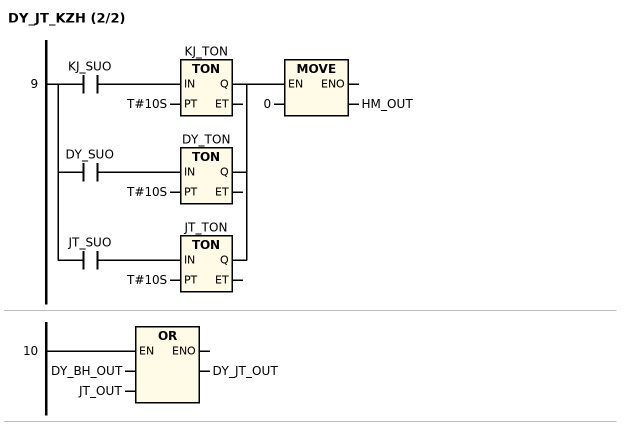
[picture p72: DY_JT_KZH (LD)]
_LD_ (* Ladder Diagram *)
NETWORK 1 (* 电源保护延时控制 *)
	{ [DY_BH_IN] | [DY_BH_OUT] } - [TD_TON_IN] - [/DY_FW] - [/JT_OUT] - [/REST] --- (DY_BH_OUT)
NETWORK 2
	[DY_BH_OUT] - [/DY_BH_IN] - DY_OPEN:YANSHI_OPEN(EN_IN: *, TIME_IN: MUL(DY_FW_SET, 60), ET_OUT => DY_BH_ET) --- (DY_FW)
NETWORK 3
	*
		EN --- LIMIT(5, DY_FW_SET, 60) => DY_FW_SET
NETWORK 4 (* 急停控制 *)
	[JT_IN] --- (JT_OUT)
NETWORK 5
	KJ_R:R_TRIG(CLK: *)
		EN --- MOVE(1) => HM_OUT
NETWORK 6
	[DY_BH_OUT] - DY_R:R_TRIG(CLK: *)
		EN --- MOVE(2) => HM_OUT
NETWORK 7
	[JT_OUT] - JT_R:R_TRIG(CLK: *)
		EN --- MOVE(4) => HM_OUT
NETWORK 8
	*
		EN --- EQ(HM_OUT, 1) => KJ_SUO
		EN --- EQ(HM_OUT, 2) => DY_SUO
		EN --- EQ(HM_OUT, 4) => JT_SUO
NETWORK 9
	{ [KJ_SUO] - KJ_TON:TON(IN: *, PT: T#10S) | [DY_SUO] - DY_TON:TON(IN: *, PT: T#10S) | [JT_SUO] - JT_TON:TON(IN: *, PT: T#10S) }
		EN --- MOVE(0) => HM_OUT
NETWORK 10
	*
		EN --- OR(DY_BH_OUT, JT_OUT) => DY_JT_OUT
_END_LD_
(* the same logic as Structured Text *)
(* Network 1: 电源保护延时控制 *)
DY_BH_OUT := (DY_BH_IN OR DY_BH_OUT) AND TD_TON_IN AND NOT DY_FW AND NOT JT_OUT AND NOT REST;
(* Network 2 *)
DY_OPEN(EN_IN := DY_BH_OUT AND NOT DY_BH_IN, TIME_IN := DY_FW_SET * 60);
DY_BH_ET := DY_OPEN.ET_OUT;
DY_FW := DY_OPEN.OUT;
(* Network 3 *)
DY_FW_SET := LIMIT(5, DY_FW_SET, 60);
(* Network 4: 急停控制 *)
JT_OUT := JT_IN;
(* Network 5 *)
KJ_R(CLK := TRUE);
IF KJ_R.Q THEN
	HM_OUT := 1;
END_IF;
(* Network 6 *)
DY_R(CLK := DY_BH_OUT);
IF DY_R.Q THEN
	HM_OUT := 2;
END_IF;
(* Network 7 *)
JT_R(CLK := JT_OUT);
IF JT_R.Q THEN
	HM_OUT := 4;
END_IF;
(* Network 8 *)
KJ_SUO := HM_OUT = 1;
DY_SUO := HM_OUT = 2;
JT_SUO := HM_OUT = 4;
(* Network 9 *)
KJ_TON(IN := KJ_SUO, PT := T#10S);
DY_TON(IN := DY_SUO, PT := T#10S);
JT_TON(IN := JT_SUO, PT := T#10S);
IF KJ_TON.Q OR DY_TON.Q OR JT_TON.Q THEN
	HM_OUT := 0;
END_IF;
(* Network 10 *)
DY_JT_OUT := DY_BH_OUT OR JT_OUT;
END_FUNCTION_BLOCK

(* POU MONI_LIANG_PW, LD *)
FUNCTION_BLOCK MONI_LIANG_PW
VAR_INPUT
	DY_IN: WORD;
	XZH_IN: INT;


	XH_IN: BOOL;


	ALA_L_T_IN: INT;
	ALA_L_T_YSH: WORD;

	ALA_H_T_IN: INT;
	ALA_H_T_YSH: WORD;


	REST: BOOL;
	JJQ_K: INT;
	JJQ_G: INT;
	YSH_IN: WORD;
END_VAR
VAR_OUTPUT
	MONI_OUT: INT;
	ALA_L_OUT: BOOL;
	ALA_H_OUT: BOOL;
	ALA_T_ET: WORD;
	PW_ZHT: WORD;
	JJQ_OUT: BOOL;
	JZ_OUT: BOOL;
END_VAR
VAR








	ALA_H_KA_0: BOOL;
	ALA_H_KA: BOOL;
	ALA_H_TON: YANSHI_OPEN;
	ALA_L_KA_0: BOOL;
	ALA_L_TON: YANSHI_OPEN;
	ALA_L_KA: BOOL;
	ALA_H_T_ET: WORD;
	ALA_L_T_ET: WORD;



	HEX_ENGIN: HEX_ENGIN;
	K1: BOOL;
	G1: BOOL;
	KJ: BOOL;
	YANSHI_OPEN: YANSHI_OPEN;
	TOF: TOF;
	YANSHI_CLOSE: YANSHI_CLOSE;
END_VAR
VAR_IN_OUT
END_VAR
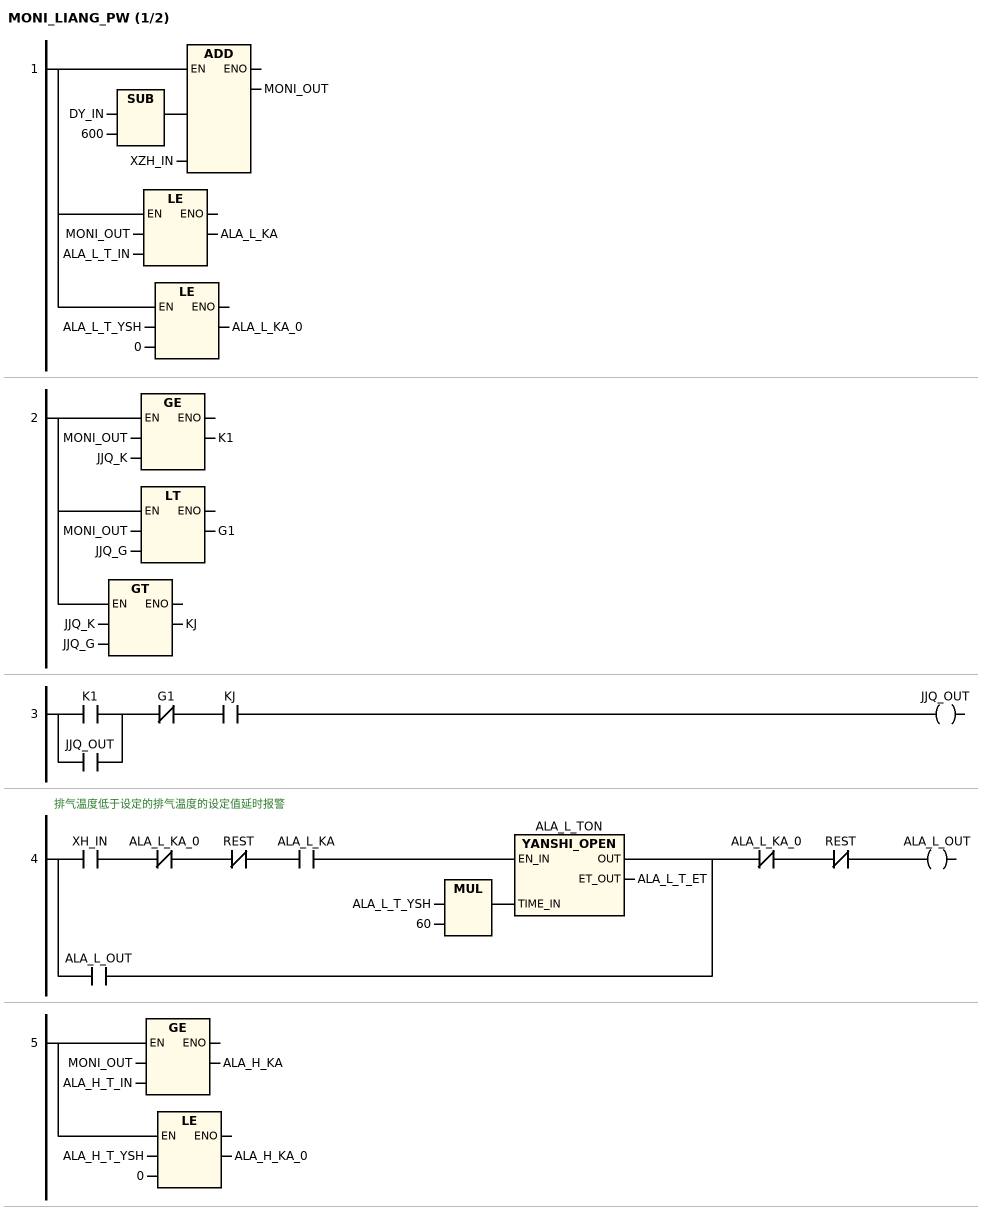
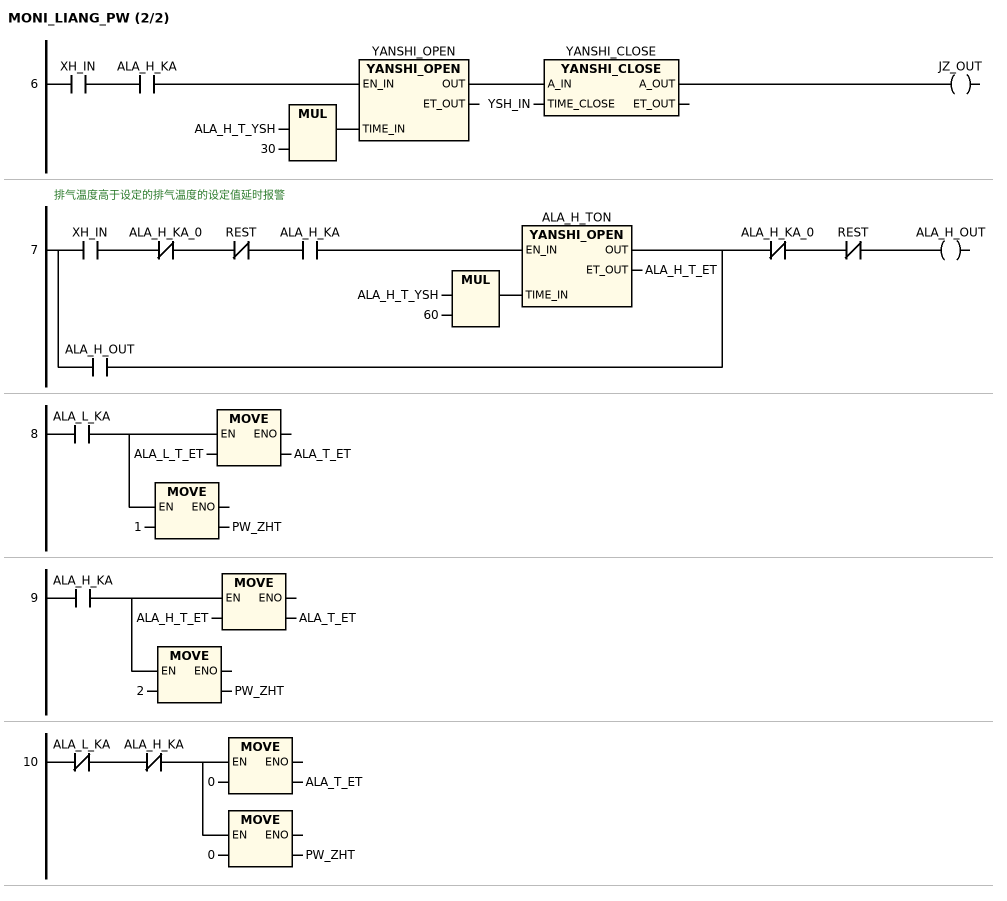
_LD_ (* Ladder Diagram *)
NETWORK 1
	*
		EN --- ADD(SUB(DY_IN, 600), XZH_IN) => MONI_OUT
		EN --- LE(MONI_OUT, ALA_L_T_IN) => ALA_L_KA
		EN --- LE(ALA_L_T_YSH, 0) => ALA_L_KA_0
NETWORK 2
	*
		EN --- GE(MONI_OUT, JJQ_K) => K1
		EN --- LT(MONI_OUT, JJQ_G) => G1
		EN --- GT(JJQ_K, JJQ_G) => KJ
NETWORK 3
	{ [K1] | [JJQ_OUT] } - [/G1] - [KJ] --- (JJQ_OUT)
NETWORK 4 (* 排气温度低于设定的排气温度的设定值延时报警 *)
	{ [XH_IN] - [/ALA_L_KA_0] - [/REST] - [ALA_L_KA] - ALA_L_TON:YANSHI_OPEN(EN_IN: *, TIME_IN: MUL(ALA_L_T_YSH, 60), ET_OUT => ALA_L_T_ET) | [ALA_L_OUT] } - [/ALA_L_KA_0] - [/REST] --- (ALA_L_OUT)
NETWORK 5
	*
		EN --- GE(MONI_OUT, ALA_H_T_IN) => ALA_H_KA
		EN --- LE(ALA_H_T_YSH, 0) => ALA_H_KA_0
NETWORK 6
	[XH_IN] - [ALA_H_KA] - YANSHI_OPEN:YANSHI_OPEN(EN_IN: *, TIME_IN: MUL(ALA_H_T_YSH, 30)) - YANSHI_CLOSE:YANSHI_CLOSE(A_IN: *, TIME_CLOSE: YSH_IN) --- (JZ_OUT)
NETWORK 7 (* 排气温度高于设定的排气温度的设定值延时报警 *)
	{ [XH_IN] - [/ALA_H_KA_0] - [/REST] - [ALA_H_KA] - ALA_H_TON:YANSHI_OPEN(EN_IN: *, TIME_IN: MUL(ALA_H_T_YSH, 60), ET_OUT => ALA_H_T_ET) | [ALA_H_OUT] } - [/ALA_H_KA_0] - [/REST] --- (ALA_H_OUT)
NETWORK 8
	[ALA_L_KA]
		EN --- MOVE(ALA_L_T_ET) => ALA_T_ET
		EN --- MOVE(1) => PW_ZHT
NETWORK 9
	[ALA_H_KA]
		EN --- MOVE(ALA_H_T_ET) => ALA_T_ET
		EN --- MOVE(2) => PW_ZHT
NETWORK 10
	[/ALA_L_KA] - [/ALA_H_KA]
		EN --- MOVE(0) => ALA_T_ET
		EN --- MOVE(0) => PW_ZHT
_END_LD_
(* the same logic as Structured Text *)
(* Network 1 *)
MONI_OUT := (DY_IN - 600) + XZH_IN;
ALA_L_KA := MONI_OUT <= ALA_L_T_IN;
ALA_L_KA_0 := ALA_L_T_YSH <= 0;
(* Network 2 *)
K1 := MONI_OUT >= JJQ_K;
G1 := MONI_OUT < JJQ_G;
KJ := JJQ_K > JJQ_G;
(* Network 3 *)
JJQ_OUT := (K1 OR JJQ_OUT) AND NOT G1 AND KJ;
(* Network 4: 排气温度低于设定的排气温度的设定值延时报警 *)
ALA_L_TON(EN_IN := XH_IN AND NOT ALA_L_KA_0 AND NOT REST AND ALA_L_KA, TIME_IN := ALA_L_T_YSH * 60);
ALA_L_T_ET := ALA_L_TON.ET_OUT;
ALA_L_OUT := (ALA_L_TON.OUT OR ALA_L_OUT) AND NOT ALA_L_KA_0 AND NOT REST;
(* Network 5 *)
ALA_H_KA := MONI_OUT >= ALA_H_T_IN;
ALA_H_KA_0 := ALA_H_T_YSH <= 0;
(* Network 6 *)
YANSHI_OPEN(EN_IN := XH_IN AND ALA_H_KA, TIME_IN := ALA_H_T_YSH * 30);
YANSHI_CLOSE(A_IN := YANSHI_OPEN.OUT, TIME_CLOSE := YSH_IN);
JZ_OUT := YANSHI_CLOSE.A_OUT;
(* Network 7: 排气温度高于设定的排气温度的设定值延时报警 *)
ALA_H_TON(EN_IN := XH_IN AND NOT ALA_H_KA_0 AND NOT REST AND ALA_H_KA, TIME_IN := ALA_H_T_YSH * 60);
ALA_H_T_ET := ALA_H_TON.ET_OUT;
ALA_H_OUT := (ALA_H_TON.OUT OR ALA_H_OUT) AND NOT ALA_H_KA_0 AND NOT REST;
(* Network 8 *)
IF ALA_L_KA THEN
	ALA_T_ET := ALA_L_T_ET;
	PW_ZHT := 1;
END_IF;
(* Network 9 *)
IF ALA_H_KA THEN
	ALA_T_ET := ALA_H_T_ET;
	PW_ZHT := 2;
END_IF;
(* Network 10 *)
IF NOT ALA_L_KA AND NOT ALA_H_KA THEN
	ALA_T_ET := 0;
	PW_ZHT := 0;
END_IF;
END_FUNCTION_BLOCK

(* POU OPEN_KJ, LD *)
FUNCTION_BLOCK OPEN_KJ
VAR_INPUT
	H_IN: WORD;
	M_IN: WORD;
	KG_IN: BOOL;
	H_OPEN_1_IN: WORD;
	M_OPEN_1_IN: WORD;
	H_CLOSE_1_IN: WORD;
       M_CLOSE_1_IN: WORD;
	H_OPEN_2_IN: WORD;
	M_OPEN_2_IN: WORD;
	H_CLOSE_2_IN: WORD;
       M_CLOSE_2_IN: WORD;
	H_OPEN_3_IN: WORD;
	M_OPEN_3_IN: WORD;
	H_CLOSE_3_IN: WORD;
       M_CLOSE_3_IN: WORD;
END_VAR
VAR_OUTPUT
	KG_OUT: BOOL;
	KZH_OUT: BOOL;
END_VAR
VAR
	OPEN_1_KA: BOOL;
	CLOSE_1_KA: BOOL;
	OPEN_2_KA: BOOL;
	CLOSE_2_KA: BOOL;
	CLOSE_3_KA: BOOL;
	OPEN_3_KA: BOOL;

	KZH_2_OUT: BOOL;
	KZH_3_OUT: BOOL;
	KZH_1_OUT: BOOL;
	AN_K: AN_NIU;
END_VAR
VAR_IN_OUT

END_VAR
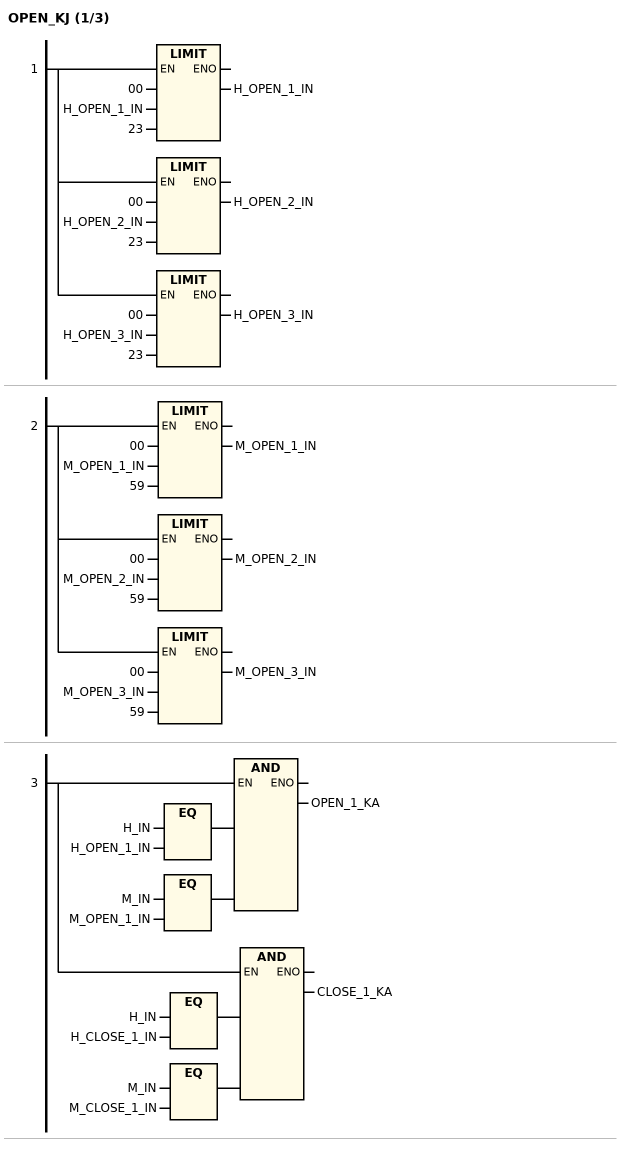
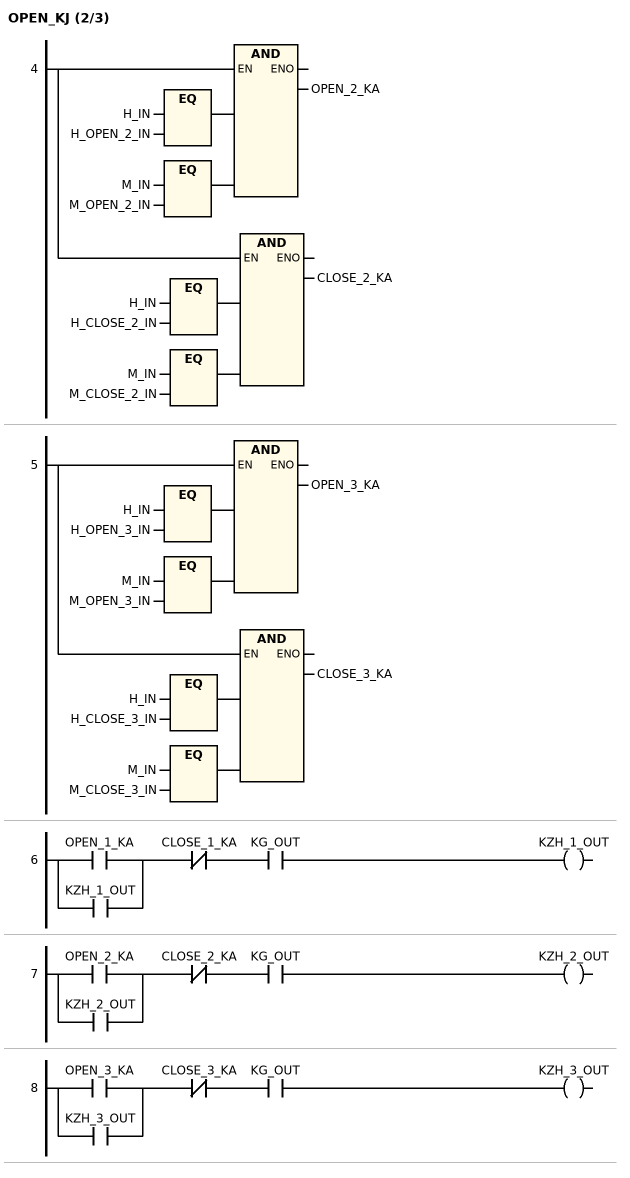
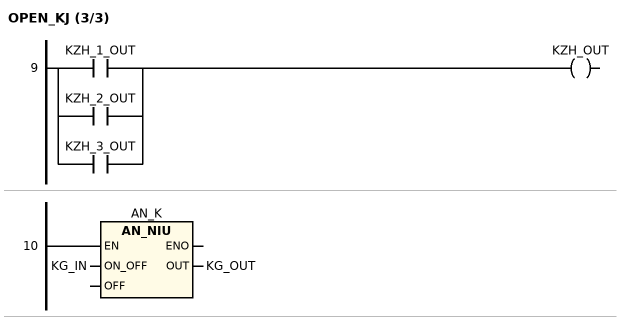
_LD_ (* Ladder Diagram *)
NETWORK 1
	*
		EN --- LIMIT(00, H_OPEN_1_IN, 23) => H_OPEN_1_IN
		EN --- LIMIT(00, H_OPEN_2_IN, 23) => H_OPEN_2_IN
		EN --- LIMIT(00, H_OPEN_3_IN, 23) => H_OPEN_3_IN
NETWORK 2
	*
		EN --- LIMIT(00, M_OPEN_1_IN, 59) => M_OPEN_1_IN
		EN --- LIMIT(00, M_OPEN_2_IN, 59) => M_OPEN_2_IN
		EN --- LIMIT(00, M_OPEN_3_IN, 59) => M_OPEN_3_IN
NETWORK 3
	*
		EN --- AND(EQ(H_IN, H_OPEN_1_IN), EQ(M_IN, M_OPEN_1_IN)) => OPEN_1_KA
		EN --- AND(EQ(H_IN, H_CLOSE_1_IN), EQ(M_IN, M_CLOSE_1_IN)) => CLOSE_1_KA
NETWORK 4
	*
		EN --- AND(EQ(H_IN, H_OPEN_2_IN), EQ(M_IN, M_OPEN_2_IN)) => OPEN_2_KA
		EN --- AND(EQ(H_IN, H_CLOSE_2_IN), EQ(M_IN, M_CLOSE_2_IN)) => CLOSE_2_KA
NETWORK 5
	*
		EN --- AND(EQ(H_IN, H_OPEN_3_IN), EQ(M_IN, M_OPEN_3_IN)) => OPEN_3_KA
		EN --- AND(EQ(H_IN, H_CLOSE_3_IN), EQ(M_IN, M_CLOSE_3_IN)) => CLOSE_3_KA
NETWORK 6
	{ [OPEN_1_KA] | [KZH_1_OUT] } - [/CLOSE_1_KA] - [KG_OUT] --- (KZH_1_OUT)
NETWORK 7
	{ [OPEN_2_KA] | [KZH_2_OUT] } - [/CLOSE_2_KA] - [KG_OUT] --- (KZH_2_OUT)
NETWORK 8
	{ [OPEN_3_KA] | [KZH_3_OUT] } - [/CLOSE_3_KA] - [KG_OUT] --- (KZH_3_OUT)
NETWORK 9
	{ [KZH_1_OUT] | [KZH_2_OUT] | [KZH_3_OUT] } --- (KZH_OUT)
NETWORK 10
	*
		EN --- AN_K:AN_NIU(ON_OFF: KG_IN, OFF: ) => KG_OUT
_END_LD_
(* the same logic as Structured Text *)
(* Network 1 *)
H_OPEN_1_IN := LIMIT(00, H_OPEN_1_IN, 23);
H_OPEN_2_IN := LIMIT(00, H_OPEN_2_IN, 23);
H_OPEN_3_IN := LIMIT(00, H_OPEN_3_IN, 23);
(* Network 2 *)
M_OPEN_1_IN := LIMIT(00, M_OPEN_1_IN, 59);
M_OPEN_2_IN := LIMIT(00, M_OPEN_2_IN, 59);
M_OPEN_3_IN := LIMIT(00, M_OPEN_3_IN, 59);
(* Network 3 *)
OPEN_1_KA := (H_IN = H_OPEN_1_IN) AND (M_IN = M_OPEN_1_IN);
CLOSE_1_KA := (H_IN = H_CLOSE_1_IN) AND (M_IN = M_CLOSE_1_IN);
(* Network 4 *)
OPEN_2_KA := (H_IN = H_OPEN_2_IN) AND (M_IN = M_OPEN_2_IN);
CLOSE_2_KA := (H_IN = H_CLOSE_2_IN) AND (M_IN = M_CLOSE_2_IN);
(* Network 5 *)
OPEN_3_KA := (H_IN = H_OPEN_3_IN) AND (M_IN = M_OPEN_3_IN);
CLOSE_3_KA := (H_IN = H_CLOSE_3_IN) AND (M_IN = M_CLOSE_3_IN);
(* Network 6 *)
KZH_1_OUT := (OPEN_1_KA OR KZH_1_OUT) AND NOT CLOSE_1_KA AND KG_OUT;
(* Network 7 *)
KZH_2_OUT := (OPEN_2_KA OR KZH_2_OUT) AND NOT CLOSE_2_KA AND KG_OUT;
(* Network 8 *)
KZH_3_OUT := (OPEN_3_KA OR KZH_3_OUT) AND NOT CLOSE_3_KA AND KG_OUT;
(* Network 9 *)
KZH_OUT := KZH_1_OUT OR KZH_2_OUT OR KZH_3_OUT;
(* Network 10: see the listing above *)
END_FUNCTION_BLOCK

(* POU DEF_YUNSUAN, LD *)
FUNCTION_BLOCK DEF_YUNSUAN
VAR_INPUT
	COOL_1_M: DWORD;
	COOL_2_M: DWORD;
	COOL_3_M: DWORD;
	COOL_4_M: DWORD;
	COOL_5_M: DWORD;
	COOL_6_M: DWORD;
	COOL_7_M: DWORD;
	COOL_8_M: DWORD;
	COOL_9_M: DWORD;
	COOL_10_M: DWORD;
	COOL_11_M: DWORD;
	COOL_12_M: DWORD;
	COOL_13_M: DWORD;
	COOL_14_M: DWORD;
	DD_1_IN: BOOL;
	DD_2_IN: BOOL;
	DD_3_IN: BOOL;
	DD_4_IN: BOOL;
	DD_5_IN: BOOL;
	DD_6_IN: BOOL;
	DD_7_IN: BOOL;
	DD_8_IN: BOOL;
	DD_9_IN: BOOL;
	DD_10_IN: BOOL;
	DD_11_IN: BOOL;
	DD_12_IN: BOOL;
	DD_13_IN: BOOL;
	DD_14_IN: BOOL;
	KSH_SET: WORD;

END_VAR
VAR_OUTPUT
	DEF_1_ZD: BOOL;
	DEF_2_ZD: BOOL;
	DEF_3_ZD: BOOL;
	DEF_4_ZD: BOOL;
	DEF_5_ZD: BOOL;
	DEF_6_ZD: BOOL;
	DEF_7_ZD: BOOL;
	DEF_8_ZD: BOOL;
	DEF_9_ZD: BOOL;
	DEF_10_ZD: BOOL;
	DEF_11_ZD: BOOL;
	DEF_12_ZD: BOOL;
	DEF_13_ZD: BOOL;
	DEF_14_ZD: BOOL;
	DEF_1_FJ: BOOL;
	DEF_2_FJ: BOOL;
	DEF_3_FJ: BOOL;
	DEF_4_FJ: BOOL;
	DEF_5_FJ: BOOL;
	DEF_6_FJ: BOOL;
	DEF_7_FJ: BOOL;
	DEF_8_FJ: BOOL;
	DEF_9_FJ: BOOL;
	DEF_10_FJ: BOOL;
	DEF_11_FJ: BOOL;
	DEF_12_FJ: BOOL;
	DEF_13_FJ: BOOL;
	DEF_14_FJ: BOOL;

END_VAR
VAR
	ROOM_1_CX: BYTE;
	ROOM_2_CX: BYTE;
	ROOM_3_CX: BYTE;
	ROOM_4_CX: BYTE;
	ROOM_5_CX: BYTE;
	ROOM_6_CX: BYTE;
	ROOM_7_CX: BYTE;
	ROOM_8_CX: BYTE;
	ROOM_9_CX: BYTE;
	ROOM_10_CX: BYTE;
	ROOM_11_CX: BYTE;
	ROOM_12_CX: BYTE;
	ROOM_13_CX: BYTE;
	ROOM_14_CX: BYTE;
	BJ_CX: BJ_MIN_DEF;
	DEF_PX: DEF_PAIXU;



	DD_1: R_TRIG;
	DD_2: R_TRIG;
	DD_3: R_TRIG;
	DD_4: R_TRIG;
	DD_5: R_TRIG;
	DD_6: R_TRIG;
	DD_7: R_TRIG;
	DD_8: R_TRIG;
	DD_9: R_TRIG;
	DD_10: R_TRIG;
	DD_11: R_TRIG;
	DD_12: R_TRIG;
	DD_13: R_TRIG;
	DD_14: R_TRIG;

END_VAR
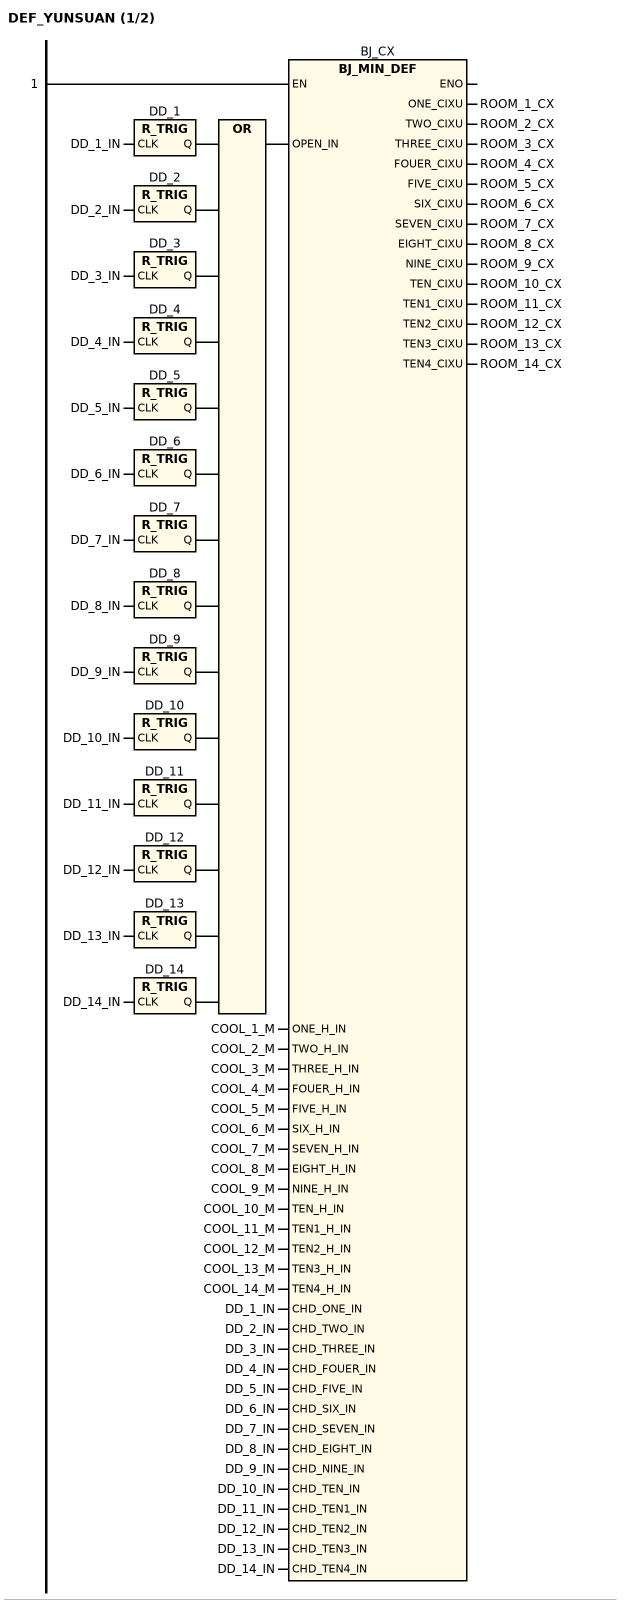
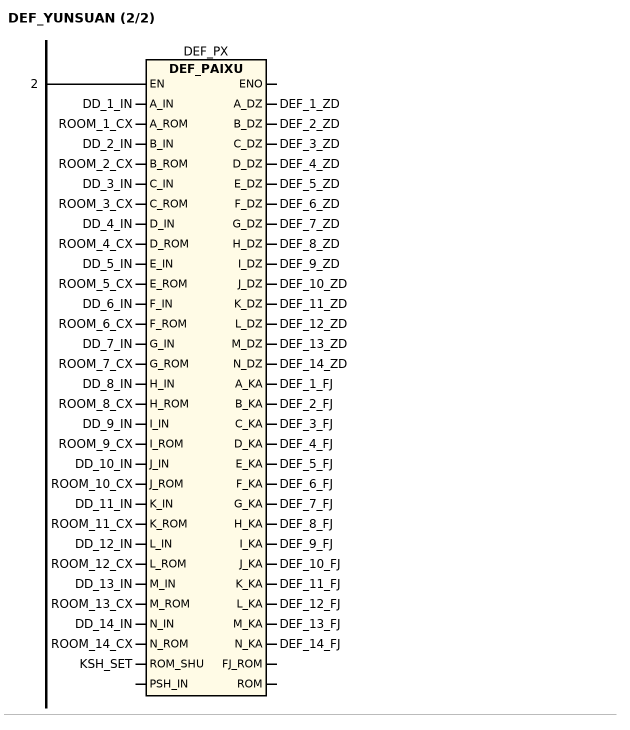
_LD_ (* Ladder Diagram *)
NETWORK 1
	*
		EN --- BJ_CX:BJ_MIN_DEF(OPEN_IN: OR(DD_1:R_TRIG(CLK: DD_1_IN), DD_2:R_TRIG(CLK: DD_2_IN), DD_3:R_TRIG(CLK: DD_3_IN), DD_4:R_TRIG(CLK: DD_4_IN), DD_5:R_TRIG(CLK: DD_5_IN), DD_6:R_TRIG(CLK: DD_6_IN), DD_7:R_TRIG(CLK: DD_7_IN), DD_8:R_TRIG(CLK: DD_8_IN), DD_9:R_TRIG(CLK: DD_9_IN), DD_10:R_TRIG(CLK: DD_10_IN), DD_11:R_TRIG(CLK: DD_11_IN), DD_12:R_TRIG(CLK: DD_12_IN), DD_13:R_TRIG(CLK: DD_13_IN), DD_14:R_TRIG(CLK: DD_14_IN)), ONE_H_IN: COOL_1_M, TWO_H_IN: COOL_2_M, THREE_H_IN: COOL_3_M, FOUER_H_IN: COOL_4_M, FIVE_H_IN: COOL_5_M, SIX_H_IN: COOL_6_M, SEVEN_H_IN: COOL_7_M, EIGHT_H_IN: COOL_8_M, NINE_H_IN: COOL_9_M, TEN_H_IN: COOL_10_M, TEN1_H_IN: COOL_11_M, TEN2_H_IN: COOL_12_M, TEN3_H_IN: COOL_13_M, TEN4_H_IN: COOL_14_M, CHD_ONE_IN: DD_1_IN, CHD_TWO_IN: DD_2_IN, CHD_THREE_IN: DD_3_IN, CHD_FOUER_IN: DD_4_IN, CHD_FIVE_IN: DD_5_IN, CHD_SIX_IN: DD_6_IN, CHD_SEVEN_IN: DD_7_IN, CHD_EIGHT_IN: DD_8_IN, CHD_NINE_IN: DD_9_IN, CHD_TEN_IN: DD_10_IN, CHD_TEN1_IN: DD_11_IN, CHD_TEN2_IN: DD_12_IN, CHD_TEN3_IN: DD_13_IN, CHD_TEN4_IN: DD_14_IN, TWO_CIXU => ROOM_2_CX, THREE_CIXU => ROOM_3_CX, FOUER_CIXU => ROOM_4_CX, FIVE_CIXU => ROOM_5_CX, SIX_CIXU => ROOM_6_CX, SEVEN_CIXU => ROOM_7_CX, EIGHT_CIXU => ROOM_8_CX, NINE_CIXU => ROOM_9_CX, TEN_CIXU => ROOM_10_CX, TEN1_CIXU => ROOM_11_CX, TEN2_CIXU => ROOM_12_CX, TEN3_CIXU => ROOM_13_CX, TEN4_CIXU => ROOM_14_CX) => ROOM_1_CX
NETWORK 2
	*
		EN --- DEF_PX:DEF_PAIXU(A_IN: DD_1_IN, A_ROM: ROOM_1_CX, B_IN: DD_2_IN, B_ROM: ROOM_2_CX, C_IN: DD_3_IN, C_ROM: ROOM_3_CX, D_IN: DD_4_IN, D_ROM: ROOM_4_CX, E_IN: DD_5_IN, E_ROM: ROOM_5_CX, F_IN: DD_6_IN, F_ROM: ROOM_6_CX, G_IN: DD_7_IN, G_ROM: ROOM_7_CX, H_IN: DD_8_IN, H_ROM: ROOM_8_CX, I_IN: DD_9_IN, I_ROM: ROOM_9_CX, J_IN: DD_10_IN, J_ROM: ROOM_10_CX, K_IN: DD_11_IN, K_ROM: ROOM_11_CX, L_IN: DD_12_IN, L_ROM: ROOM_12_CX, M_IN: DD_13_IN, M_ROM: ROOM_13_CX, N_IN: DD_14_IN, N_ROM: ROOM_14_CX, ROM_SHU: KSH_SET, PSH_IN: , B_DZ => DEF_2_ZD, C_DZ => DEF_3_ZD, D_DZ => DEF_4_ZD, E_DZ => DEF_5_ZD, F_DZ => DEF_6_ZD, G_DZ => DEF_7_ZD, H_DZ => DEF_8_ZD, I_DZ => DEF_9_ZD, J_DZ => DEF_10_ZD, K_DZ => DEF_11_ZD, L_DZ => DEF_12_ZD, M_DZ => DEF_13_ZD, N_DZ => DEF_14_ZD, A_KA => DEF_1_FJ, B_KA => DEF_2_FJ, C_KA => DEF_3_FJ, D_KA => DEF_4_FJ, E_KA => DEF_5_FJ, F_KA => DEF_6_FJ, G_KA => DEF_7_FJ, H_KA => DEF_8_FJ, I_KA => DEF_9_FJ, J_KA => DEF_10_FJ, K_KA => DEF_11_FJ, L_KA => DEF_12_FJ, M_KA => DEF_13_FJ, N_KA => DEF_14_FJ) => DEF_1_ZD
_END_LD_
(* the same logic as Structured Text *)
(* Network 1 *)
DD_1(CLK := DD_1_IN);
DD_2(CLK := DD_2_IN);
DD_3(CLK := DD_3_IN);
DD_4(CLK := DD_4_IN);
DD_5(CLK := DD_5_IN);
DD_6(CLK := DD_6_IN);
DD_7(CLK := DD_7_IN);
DD_8(CLK := DD_8_IN);
DD_9(CLK := DD_9_IN);
DD_10(CLK := DD_10_IN);
DD_11(CLK := DD_11_IN);
DD_12(CLK := DD_12_IN);
DD_13(CLK := DD_13_IN);
DD_14(CLK := DD_14_IN);
BJ_CX(OPEN_IN := DD_1.Q OR DD_2.Q OR DD_3.Q OR DD_4.Q OR DD_5.Q OR DD_6.Q OR DD_7.Q OR DD_8.Q OR DD_9.Q OR DD_10.Q OR DD_11.Q OR DD_12.Q OR DD_13.Q OR DD_14.Q, ONE_H_IN := COOL_1_M, TWO_H_IN := COOL_2_M, THREE_H_IN := COOL_3_M, FOUER_H_IN := COOL_4_M, FIVE_H_IN := COOL_5_M, SIX_H_IN := COOL_6_M, SEVEN_H_IN := COOL_7_M, EIGHT_H_IN := COOL_8_M, NINE_H_IN := COOL_9_M, TEN_H_IN := COOL_10_M, TEN1_H_IN := COOL_11_M, TEN2_H_IN := COOL_12_M, TEN3_H_IN := COOL_13_M, TEN4_H_IN := COOL_14_M, CHD_ONE_IN := DD_1_IN, CHD_TWO_IN := DD_2_IN, CHD_THREE_IN := DD_3_IN, CHD_FOUER_IN := DD_4_IN, CHD_FIVE_IN := DD_5_IN, CHD_SIX_IN := DD_6_IN, CHD_SEVEN_IN := DD_7_IN, CHD_EIGHT_IN := DD_8_IN, CHD_NINE_IN := DD_9_IN, CHD_TEN_IN := DD_10_IN, CHD_TEN1_IN := DD_11_IN, CHD_TEN2_IN := DD_12_IN, CHD_TEN3_IN := DD_13_IN, CHD_TEN4_IN := DD_14_IN);
ROOM_2_CX := BJ_CX.TWO_CIXU;
ROOM_3_CX := BJ_CX.THREE_CIXU;
ROOM_4_CX := BJ_CX.FOUER_CIXU;
ROOM_5_CX := BJ_CX.FIVE_CIXU;
ROOM_6_CX := BJ_CX.SIX_CIXU;
ROOM_7_CX := BJ_CX.SEVEN_CIXU;
ROOM_8_CX := BJ_CX.EIGHT_CIXU;
ROOM_9_CX := BJ_CX.NINE_CIXU;
ROOM_10_CX := BJ_CX.TEN_CIXU;
ROOM_11_CX := BJ_CX.TEN1_CIXU;
ROOM_12_CX := BJ_CX.TEN2_CIXU;
ROOM_13_CX := BJ_CX.TEN3_CIXU;
ROOM_14_CX := BJ_CX.TEN4_CIXU;
ROOM_1_CX := BJ_CX.ONE_CIXU;
(* Network 2: see the listing above *)
END_FUNCTION_BLOCK

(* POU BJ_MIN_DEF, LD *)
FUNCTION_BLOCK BJ_MIN_DEF
VAR_INPUT
	OPEN_IN: BOOL;
	ONE_H_IN: DWORD;
	TWO_H_IN: DWORD;
	THREE_H_IN: DWORD;
	FOUER_H_IN: DWORD;
	FIVE_H_IN: DWORD;
	SIX_H_IN: DWORD;
	SEVEN_H_IN: DWORD;
	EIGHT_H_IN: DWORD;
	NINE_H_IN: DWORD;
	TEN_H_IN: DWORD;
	TEN1_H_IN: DWORD;
	TEN2_H_IN: DWORD;
	TEN3_H_IN: DWORD;
	TEN4_H_IN: DWORD;
	CHD_ONE_IN: BOOL;
	CHD_TWO_IN: BOOL;
	CHD_THREE_IN: BOOL;
	CHD_FOUER_IN: BOOL;
	CHD_FIVE_IN: BOOL;
	CHD_SIX_IN: BOOL;
	CHD_SEVEN_IN: BOOL;
	CHD_EIGHT_IN: BOOL;
	CHD_NINE_IN: BOOL;
	CHD_TEN_IN: BOOL;
	CHD_TEN1_IN: BOOL;
	CHD_TEN2_IN: BOOL;
	CHD_TEN3_IN: BOOL;
	CHD_TEN4_IN: BOOL;

END_VAR
VAR_OUTPUT
	ONE_CIXU: BYTE;
	TWO_CIXU: BYTE;
	THREE_CIXU: BYTE;
	FOUER_CIXU: BYTE;
	FIVE_CIXU: BYTE;
	SIX_CIXU: BYTE;
	SEVEN_CIXU: BYTE;
	EIGHT_CIXU: BYTE;
	NINE_CIXU: BYTE;
	TEN_CIXU: BYTE;
	TEN1_CIXU: BYTE;
	TEN2_CIXU: BYTE;
	TEN3_CIXU: BYTE;
	TEN4_CIXU: BYTE;
END_VAR
VAR
	ONE_H_ZC_1: DWORD;
	TWO_H_ZC_1: DWORD;
	THREE_H_ZC_1: DWORD;
	FOUER_H_ZC_1: DWORD;
	FIVE_H_ZC_1: DWORD;
	ONE_CX_ZC: BYTE;
	TWO_CX_ZC: BYTE;
	THREE_CX_ZC: BYTE;
	FOUER_CX_ZC: BYTE;
	FIVE_CX_ZC: BYTE;
	ONE_H_ZC_2: DWORD;
	TWO_H_ZC_2: DWORD;
	THREE_H_ZC_2: DWORD;
	FOUER_H_ZC_2: DWORD;
	FIVE_H_ZC_2: DWORD;
	ONE_FUWEI: BOOL;
	TWO_FUWEI: BOOL;
	FIVE_FUWEI: BOOL;
	FOUER_FUWEI: BOOL;
	THREE_FUWEI: BOOL;
	EIGHT_H_ZC_1: DWORD;
	SEVEN_H_ZC_1: DWORD;
	SIX_H_ZC_1: DWORD;
	SIX_CX_ZC: BYTE;
	SEVEN_CX_ZC: BYTE;
	EIGHT_CX_ZC: BYTE;
	SIX_FUWEI: BOOL;
	SEVEN_FUWEI: BOOL;
	EIGHT_FUWEI: BOOL;
	SEVEN_H_ZC_2: DWORD;
	EIGHT_H_ZC_2: DWORD;
	NINE_H_ZC_2: DWORD;
	TEN_H_ZC_2: DWORD;
	SIX_H_ZC_2: DWORD;
	NINE_H_ZC_1: DWORD;
	TEN_H_ZC_1: DWORD;
	NINE_CX_ZC: BYTE;
	TEN_CX_ZC: BYTE;
	TEN_FUWEI: BOOL;
	NINE_FUWEI: BOOL;
	CIXU_BJ: BJ_CIXU_DEF;
	TEN1_H_ZC_1: DWORD;
	TEN2_H_ZC_1: DWORD;
	TEN3_H_ZC_1: DWORD;
	TEN4_H_ZC_1: DWORD;
	TEN1_FUWEI: BOOL;
	TEN2_FUWEI: BOOL;
	TEN3_FUWEI: BOOL;
	TEN4_FUWEI: BOOL;
	TEN1_H_ZC_2: DWORD;
	TEN2_H_ZC_2: DWORD;
	TEN3_H_ZC_2: DWORD;
	TEN4_H_ZC_2: DWORD;
	TEN4_CX_ZC: BYTE;
	TEN3_CX_ZC: BYTE;
	TEN2_CX_ZC: BYTE;
	TEN1_CX_ZC: BYTE;
END_VAR
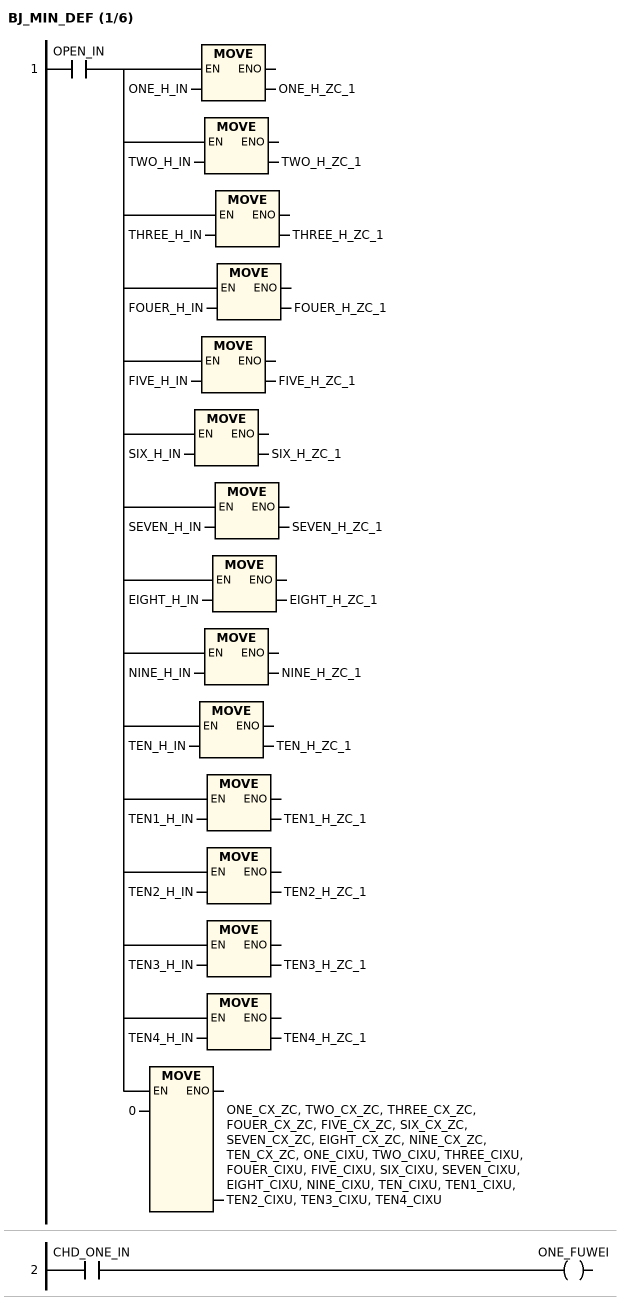
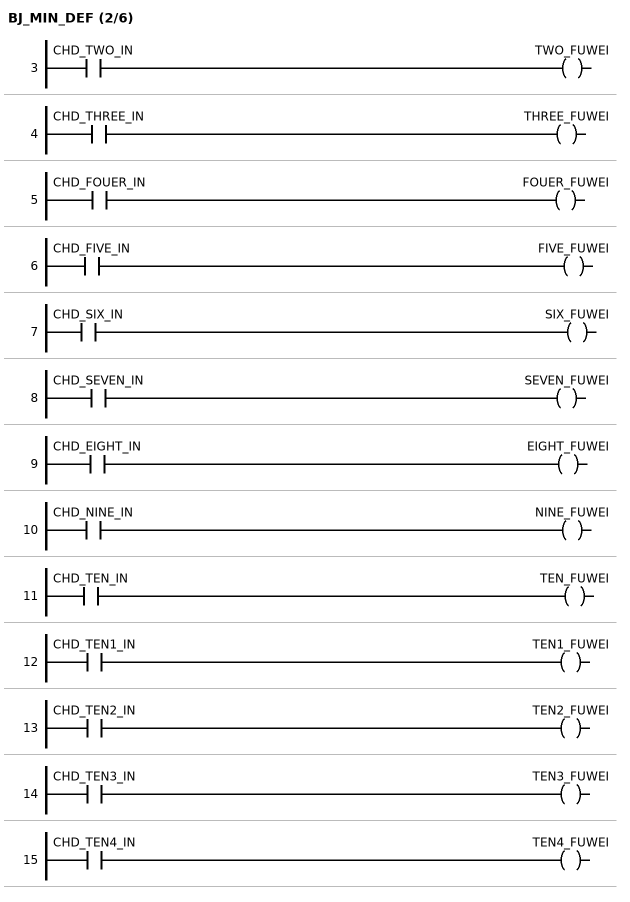
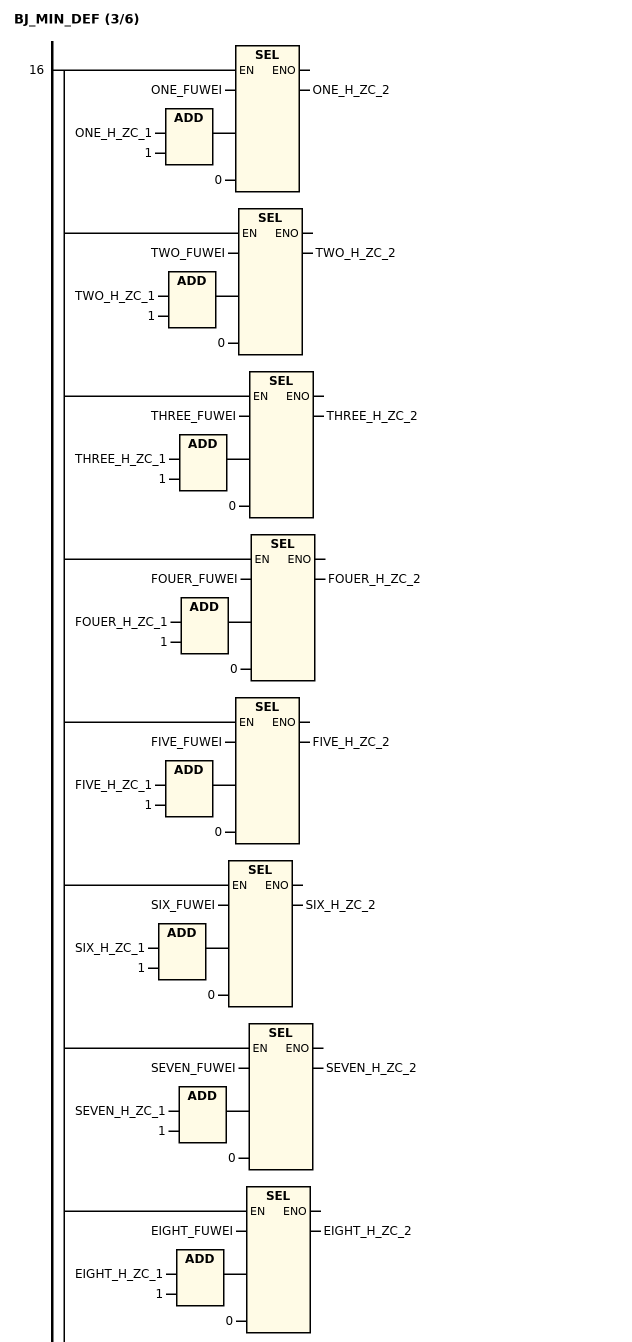
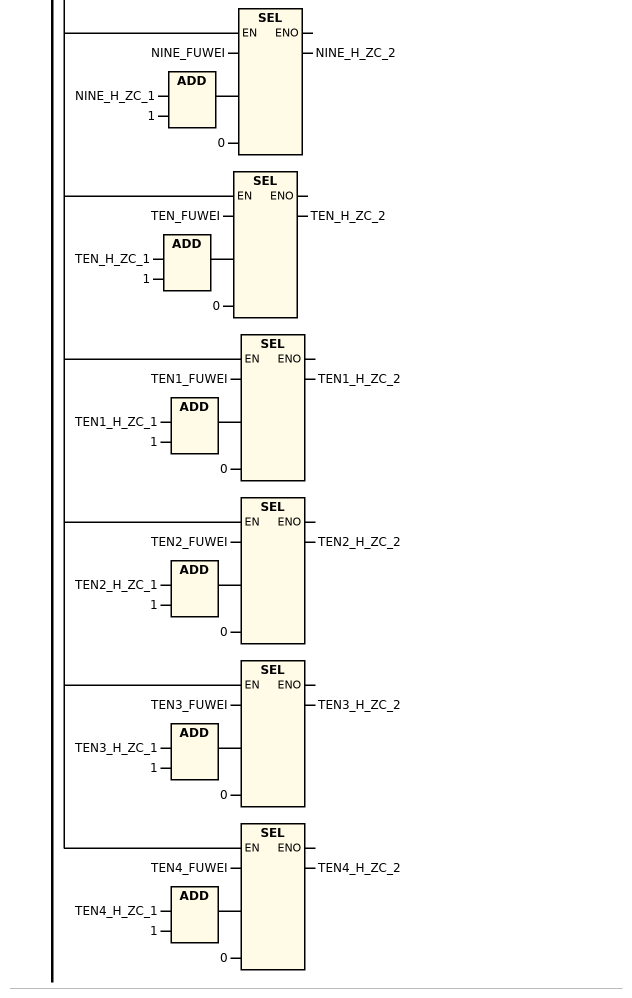
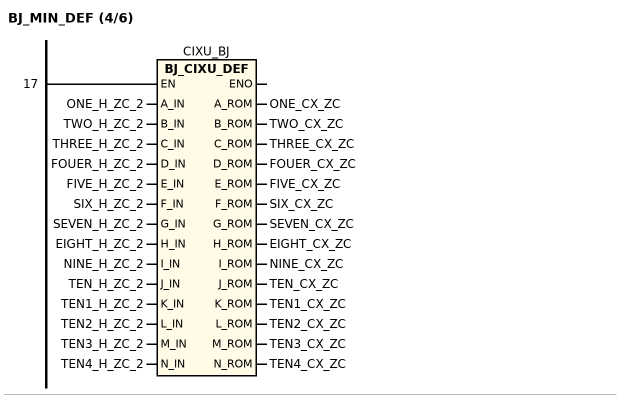
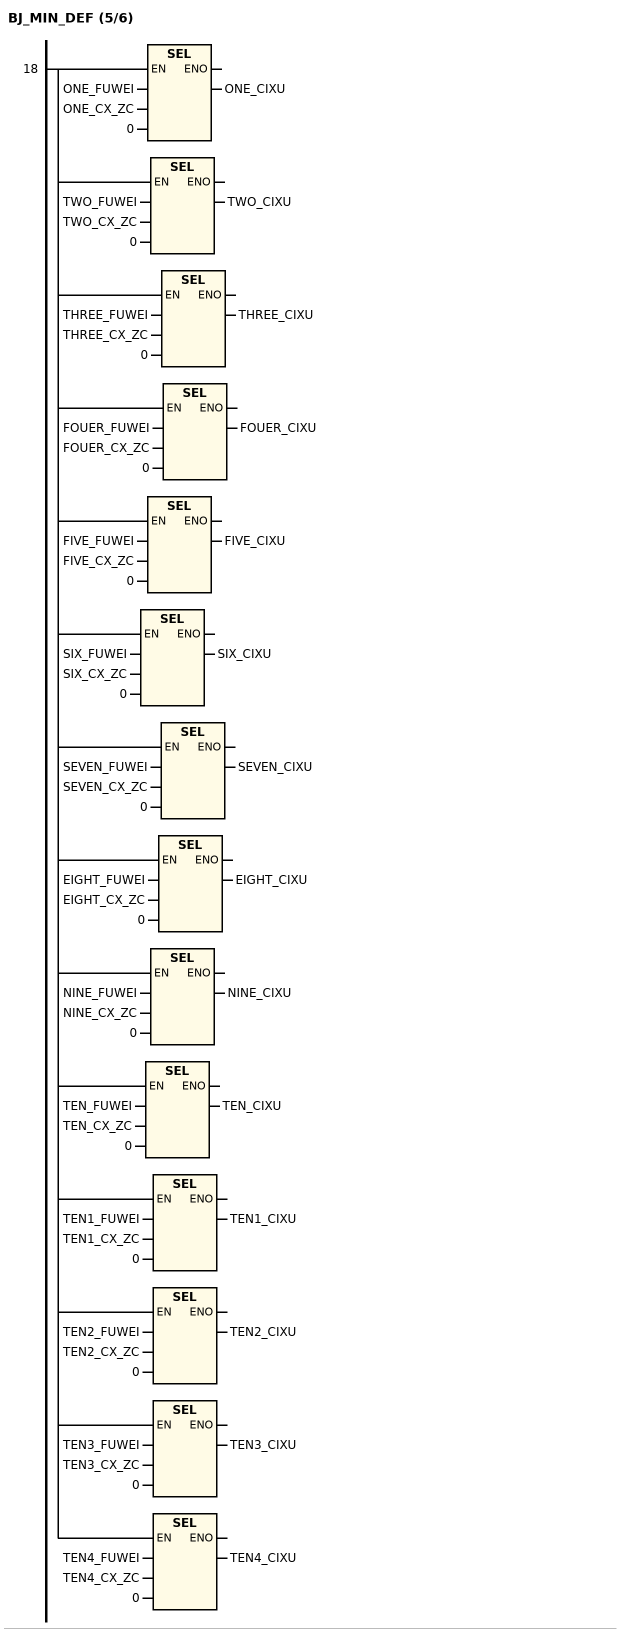
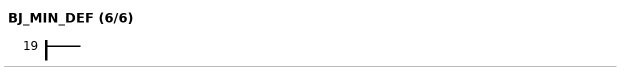
_LD_ (* Ladder Diagram *)
NETWORK 1
	[OPEN_IN]
		EN --- MOVE(ONE_H_IN) => ONE_H_ZC_1
		EN --- MOVE(TWO_H_IN) => TWO_H_ZC_1
		EN --- MOVE(THREE_H_IN) => THREE_H_ZC_1
		EN --- MOVE(FOUER_H_IN) => FOUER_H_ZC_1
		EN --- MOVE(FIVE_H_IN) => FIVE_H_ZC_1
		EN --- MOVE(SIX_H_IN) => SIX_H_ZC_1
		EN --- MOVE(SEVEN_H_IN) => SEVEN_H_ZC_1
		EN --- MOVE(EIGHT_H_IN) => EIGHT_H_ZC_1
		EN --- MOVE(NINE_H_IN) => NINE_H_ZC_1
		EN --- MOVE(TEN_H_IN) => TEN_H_ZC_1
		EN --- MOVE(TEN1_H_IN) => TEN1_H_ZC_1
		EN --- MOVE(TEN2_H_IN) => TEN2_H_ZC_1
		EN --- MOVE(TEN3_H_IN) => TEN3_H_ZC_1
		EN --- MOVE(TEN4_H_IN) => TEN4_H_ZC_1
		EN --- MOVE(0) => ONE_CX_ZC, TWO_CX_ZC, THREE_CX_ZC, FOUER_CX_ZC, FIVE_CX_ZC, SIX_CX_ZC, SEVEN_CX_ZC, EIGHT_CX_ZC, NINE_CX_ZC, TEN_CX_ZC, ONE_CIXU, TWO_CIXU, THREE_CIXU, FOUER_CIXU, FIVE_CIXU, SIX_CIXU, SEVEN_CIXU, EIGHT_CIXU, NINE_CIXU, TEN_CIXU, TEN1_CIXU, TEN2_CIXU, TEN3_CIXU, TEN4_CIXU
NETWORK 2
	[CHD_ONE_IN] --- (ONE_FUWEI)
NETWORK 3
	[CHD_TWO_IN] --- (TWO_FUWEI)
NETWORK 4
	[CHD_THREE_IN] --- (THREE_FUWEI)
NETWORK 5
	[CHD_FOUER_IN] --- (FOUER_FUWEI)
NETWORK 6
	[CHD_FIVE_IN] --- (FIVE_FUWEI)
NETWORK 7
	[CHD_SIX_IN] --- (SIX_FUWEI)
NETWORK 8
	[CHD_SEVEN_IN] --- (SEVEN_FUWEI)
NETWORK 9
	[CHD_EIGHT_IN] --- (EIGHT_FUWEI)
NETWORK 10
	[CHD_NINE_IN] --- (NINE_FUWEI)
NETWORK 11
	[CHD_TEN_IN] --- (TEN_FUWEI)
NETWORK 12
	[CHD_TEN1_IN] --- (TEN1_FUWEI)
NETWORK 13
	[CHD_TEN2_IN] --- (TEN2_FUWEI)
NETWORK 14
	[CHD_TEN3_IN] --- (TEN3_FUWEI)
NETWORK 15
	[CHD_TEN4_IN] --- (TEN4_FUWEI)
NETWORK 16
	*
		EN --- SEL(ONE_FUWEI, ADD(ONE_H_ZC_1, 1), 0) => ONE_H_ZC_2
		EN --- SEL(TWO_FUWEI, ADD(TWO_H_ZC_1, 1), 0) => TWO_H_ZC_2
		EN --- SEL(THREE_FUWEI, ADD(THREE_H_ZC_1, 1), 0) => THREE_H_ZC_2
		EN --- SEL(FOUER_FUWEI, ADD(FOUER_H_ZC_1, 1), 0) => FOUER_H_ZC_2
		EN --- SEL(FIVE_FUWEI, ADD(FIVE_H_ZC_1, 1), 0) => FIVE_H_ZC_2
		EN --- SEL(SIX_FUWEI, ADD(SIX_H_ZC_1, 1), 0) => SIX_H_ZC_2
		EN --- SEL(SEVEN_FUWEI, ADD(SEVEN_H_ZC_1, 1), 0) => SEVEN_H_ZC_2
		EN --- SEL(EIGHT_FUWEI, ADD(EIGHT_H_ZC_1, 1), 0) => EIGHT_H_ZC_2
		EN --- SEL(NINE_FUWEI, ADD(NINE_H_ZC_1, 1), 0) => NINE_H_ZC_2
		EN --- SEL(TEN_FUWEI, ADD(TEN_H_ZC_1, 1), 0) => TEN_H_ZC_2
		EN --- SEL(TEN1_FUWEI, ADD(TEN1_H_ZC_1, 1), 0) => TEN1_H_ZC_2
		EN --- SEL(TEN2_FUWEI, ADD(TEN2_H_ZC_1, 1), 0) => TEN2_H_ZC_2
		EN --- SEL(TEN3_FUWEI, ADD(TEN3_H_ZC_1, 1), 0) => TEN3_H_ZC_2
		EN --- SEL(TEN4_FUWEI, ADD(TEN4_H_ZC_1, 1), 0) => TEN4_H_ZC_2
NETWORK 17
	*
		EN --- CIXU_BJ:BJ_CIXU_DEF(A_IN: ONE_H_ZC_2, B_IN: TWO_H_ZC_2, C_IN: THREE_H_ZC_2, D_IN: FOUER_H_ZC_2, E_IN: FIVE_H_ZC_2, F_IN: SIX_H_ZC_2, G_IN: SEVEN_H_ZC_2, H_IN: EIGHT_H_ZC_2, I_IN: NINE_H_ZC_2, J_IN: TEN_H_ZC_2, K_IN: TEN1_H_ZC_2, L_IN: TEN2_H_ZC_2, M_IN: TEN3_H_ZC_2, N_IN: TEN4_H_ZC_2, B_ROM => TWO_CX_ZC, C_ROM => THREE_CX_ZC, D_ROM => FOUER_CX_ZC, E_ROM => FIVE_CX_ZC, F_ROM => SIX_CX_ZC, G_ROM => SEVEN_CX_ZC, H_ROM => EIGHT_CX_ZC, I_ROM => NINE_CX_ZC, J_ROM => TEN_CX_ZC, K_ROM => TEN1_CX_ZC, L_ROM => TEN2_CX_ZC, M_ROM => TEN3_CX_ZC, N_ROM => TEN4_CX_ZC) => ONE_CX_ZC
NETWORK 18
	*
		EN --- SEL(ONE_FUWEI, ONE_CX_ZC, 0) => ONE_CIXU
		EN --- SEL(TWO_FUWEI, TWO_CX_ZC, 0) => TWO_CIXU
		EN --- SEL(THREE_FUWEI, THREE_CX_ZC, 0) => THREE_CIXU
		EN --- SEL(FOUER_FUWEI, FOUER_CX_ZC, 0) => FOUER_CIXU
		EN --- SEL(FIVE_FUWEI, FIVE_CX_ZC, 0) => FIVE_CIXU
		EN --- SEL(SIX_FUWEI, SIX_CX_ZC, 0) => SIX_CIXU
		EN --- SEL(SEVEN_FUWEI, SEVEN_CX_ZC, 0) => SEVEN_CIXU
		EN --- SEL(EIGHT_FUWEI, EIGHT_CX_ZC, 0) => EIGHT_CIXU
		EN --- SEL(NINE_FUWEI, NINE_CX_ZC, 0) => NINE_CIXU
		EN --- SEL(TEN_FUWEI, TEN_CX_ZC, 0) => TEN_CIXU
		EN --- SEL(TEN1_FUWEI, TEN1_CX_ZC, 0) => TEN1_CIXU
		EN --- SEL(TEN2_FUWEI, TEN2_CX_ZC, 0) => TEN2_CIXU
		EN --- SEL(TEN3_FUWEI, TEN3_CX_ZC, 0) => TEN3_CIXU
		EN --- SEL(TEN4_FUWEI, TEN4_CX_ZC, 0) => TEN4_CIXU
NETWORK 19
	*
_END_LD_
(* the same logic as Structured Text *)
(* Network 1: see the listing above *)
(* Network 2 *)
ONE_FUWEI := CHD_ONE_IN;
(* Network 3 *)
TWO_FUWEI := CHD_TWO_IN;
(* Network 4 *)
THREE_FUWEI := CHD_THREE_IN;
(* Network 5 *)
FOUER_FUWEI := CHD_FOUER_IN;
(* Network 6 *)
FIVE_FUWEI := CHD_FIVE_IN;
(* Network 7 *)
SIX_FUWEI := CHD_SIX_IN;
(* Network 8 *)
SEVEN_FUWEI := CHD_SEVEN_IN;
(* Network 9 *)
EIGHT_FUWEI := CHD_EIGHT_IN;
(* Network 10 *)
NINE_FUWEI := CHD_NINE_IN;
(* Network 11 *)
TEN_FUWEI := CHD_TEN_IN;
(* Network 12 *)
TEN1_FUWEI := CHD_TEN1_IN;
(* Network 13 *)
TEN2_FUWEI := CHD_TEN2_IN;
(* Network 14 *)
TEN3_FUWEI := CHD_TEN3_IN;
(* Network 15 *)
TEN4_FUWEI := CHD_TEN4_IN;
(* Network 16 *)
ONE_H_ZC_2 := SEL(ONE_FUWEI, ONE_H_ZC_1 + 1, 0);
TWO_H_ZC_2 := SEL(TWO_FUWEI, TWO_H_ZC_1 + 1, 0);
THREE_H_ZC_2 := SEL(THREE_FUWEI, THREE_H_ZC_1 + 1, 0);
FOUER_H_ZC_2 := SEL(FOUER_FUWEI, FOUER_H_ZC_1 + 1, 0);
FIVE_H_ZC_2 := SEL(FIVE_FUWEI, FIVE_H_ZC_1 + 1, 0);
SIX_H_ZC_2 := SEL(SIX_FUWEI, SIX_H_ZC_1 + 1, 0);
SEVEN_H_ZC_2 := SEL(SEVEN_FUWEI, SEVEN_H_ZC_1 + 1, 0);
EIGHT_H_ZC_2 := SEL(EIGHT_FUWEI, EIGHT_H_ZC_1 + 1, 0);
NINE_H_ZC_2 := SEL(NINE_FUWEI, NINE_H_ZC_1 + 1, 0);
TEN_H_ZC_2 := SEL(TEN_FUWEI, TEN_H_ZC_1 + 1, 0);
TEN1_H_ZC_2 := SEL(TEN1_FUWEI, TEN1_H_ZC_1 + 1, 0);
TEN2_H_ZC_2 := SEL(TEN2_FUWEI, TEN2_H_ZC_1 + 1, 0);
TEN3_H_ZC_2 := SEL(TEN3_FUWEI, TEN3_H_ZC_1 + 1, 0);
TEN4_H_ZC_2 := SEL(TEN4_FUWEI, TEN4_H_ZC_1 + 1, 0);
(* Network 17 *)
CIXU_BJ(A_IN := ONE_H_ZC_2, B_IN := TWO_H_ZC_2, C_IN := THREE_H_ZC_2, D_IN := FOUER_H_ZC_2, E_IN := FIVE_H_ZC_2, F_IN := SIX_H_ZC_2, G_IN := SEVEN_H_ZC_2, H_IN := EIGHT_H_ZC_2, I_IN := NINE_H_ZC_2, J_IN := TEN_H_ZC_2, K_IN := TEN1_H_ZC_2, L_IN := TEN2_H_ZC_2, M_IN := TEN3_H_ZC_2, N_IN := TEN4_H_ZC_2);
TWO_CX_ZC := CIXU_BJ.B_ROM;
THREE_CX_ZC := CIXU_BJ.C_ROM;
FOUER_CX_ZC := CIXU_BJ.D_ROM;
FIVE_CX_ZC := CIXU_BJ.E_ROM;
SIX_CX_ZC := CIXU_BJ.F_ROM;
SEVEN_CX_ZC := CIXU_BJ.G_ROM;
EIGHT_CX_ZC := CIXU_BJ.H_ROM;
NINE_CX_ZC := CIXU_BJ.I_ROM;
TEN_CX_ZC := CIXU_BJ.J_ROM;
TEN1_CX_ZC := CIXU_BJ.K_ROM;
TEN2_CX_ZC := CIXU_BJ.L_ROM;
TEN3_CX_ZC := CIXU_BJ.M_ROM;
TEN4_CX_ZC := CIXU_BJ.N_ROM;
ONE_CX_ZC := CIXU_BJ.A_ROM;
(* Network 18 *)
ONE_CIXU := SEL(ONE_FUWEI, ONE_CX_ZC, 0);
TWO_CIXU := SEL(TWO_FUWEI, TWO_CX_ZC, 0);
THREE_CIXU := SEL(THREE_FUWEI, THREE_CX_ZC, 0);
FOUER_CIXU := SEL(FOUER_FUWEI, FOUER_CX_ZC, 0);
FIVE_CIXU := SEL(FIVE_FUWEI, FIVE_CX_ZC, 0);
SIX_CIXU := SEL(SIX_FUWEI, SIX_CX_ZC, 0);
SEVEN_CIXU := SEL(SEVEN_FUWEI, SEVEN_CX_ZC, 0);
EIGHT_CIXU := SEL(EIGHT_FUWEI, EIGHT_CX_ZC, 0);
NINE_CIXU := SEL(NINE_FUWEI, NINE_CX_ZC, 0);
TEN_CIXU := SEL(TEN_FUWEI, TEN_CX_ZC, 0);
TEN1_CIXU := SEL(TEN1_FUWEI, TEN1_CX_ZC, 0);
TEN2_CIXU := SEL(TEN2_FUWEI, TEN2_CX_ZC, 0);
TEN3_CIXU := SEL(TEN3_FUWEI, TEN3_CX_ZC, 0);
TEN4_CIXU := SEL(TEN4_FUWEI, TEN4_CX_ZC, 0);
(* Network 19: see the listing above *)
END_FUNCTION_BLOCK

(* POU BJ_CIXU_DEF, LD *)
FUNCTION_BLOCK BJ_CIXU_DEF
VAR_INPUT
	A_IN:DWORD;
	B_IN: DWORD;
	C_IN: DWORD;
	D_IN: DWORD;
	E_IN: DWORD;
	F_IN: DWORD;
	G_IN: DWORD;
	H_IN: DWORD;
	I_IN: DWORD;
	J_IN: DWORD;
	K_IN: DWORD;
	L_IN: DWORD;
	M_IN: DWORD;
	N_IN: DWORD;
END_VAR
VAR_OUTPUT
	A_ROM: BYTE;
	B_ROM: BYTE;
	C_ROM: BYTE;
	D_ROM: BYTE;
	E_ROM: BYTE;
	F_ROM: BYTE;
	G_ROM: BYTE;
	H_ROM: BYTE;
	I_ROM: BYTE;
	J_ROM: BYTE;
	K_ROM: BYTE;
	L_ROM: BYTE;
	M_ROM: BYTE;
	N_ROM: BYTE;
END_VAR
VAR
END_VAR
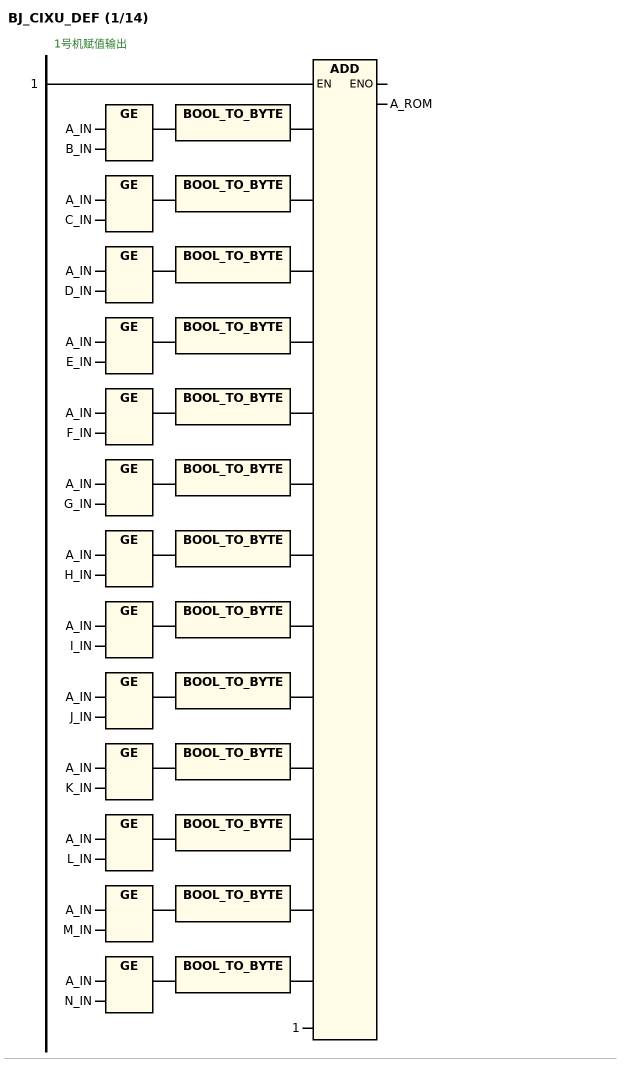
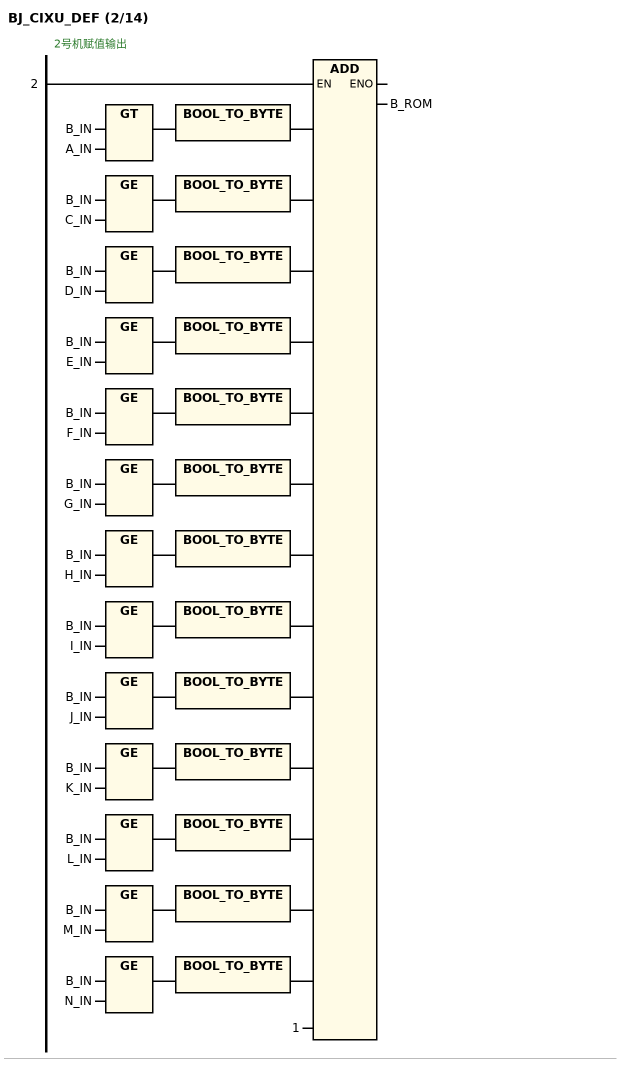
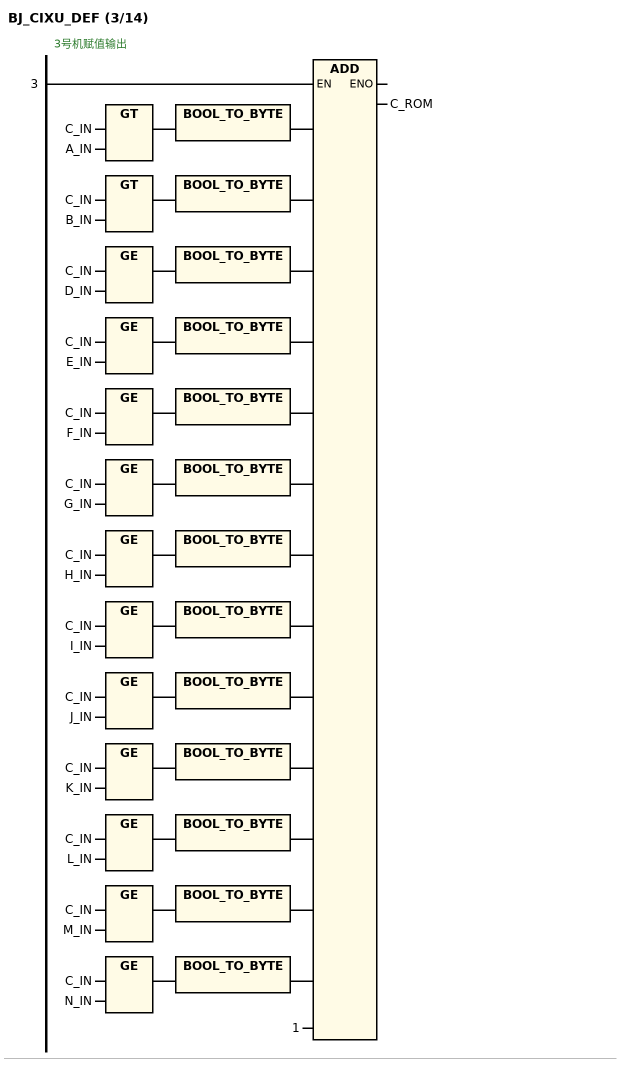
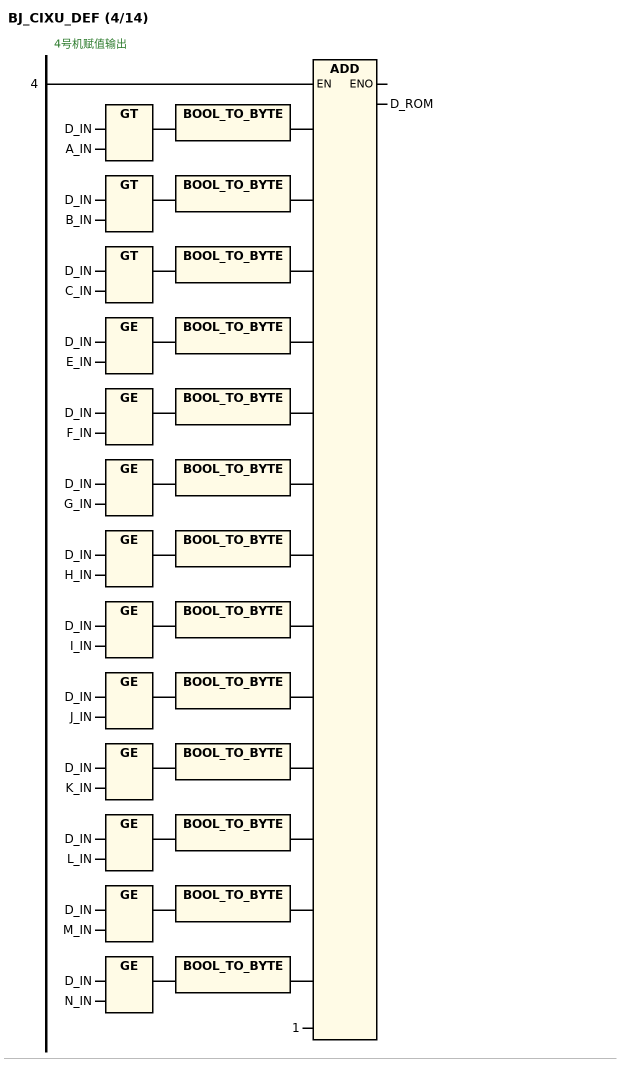
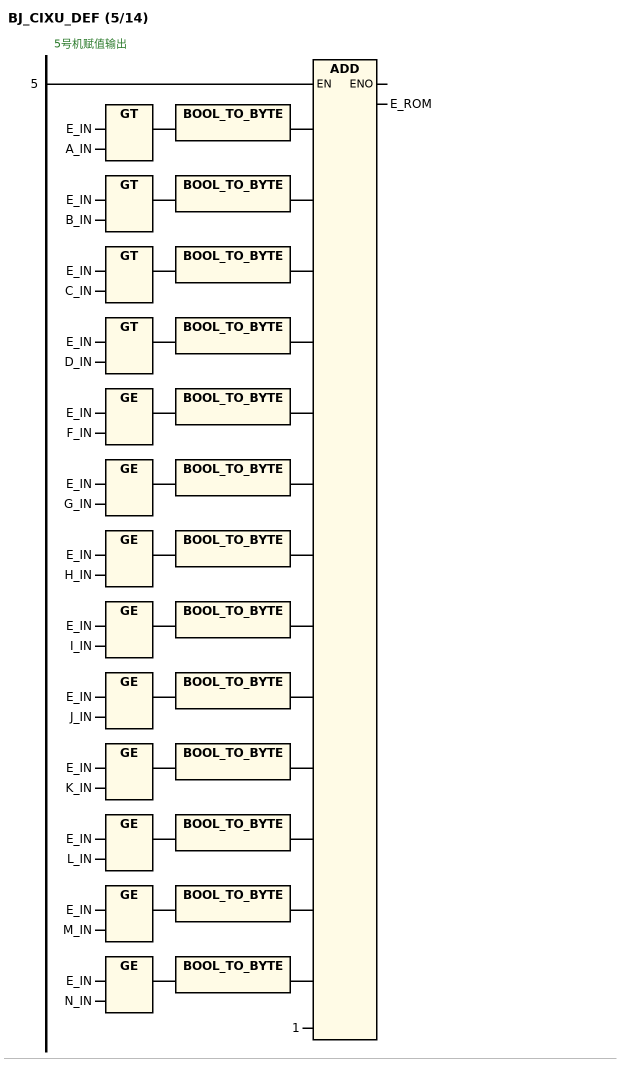
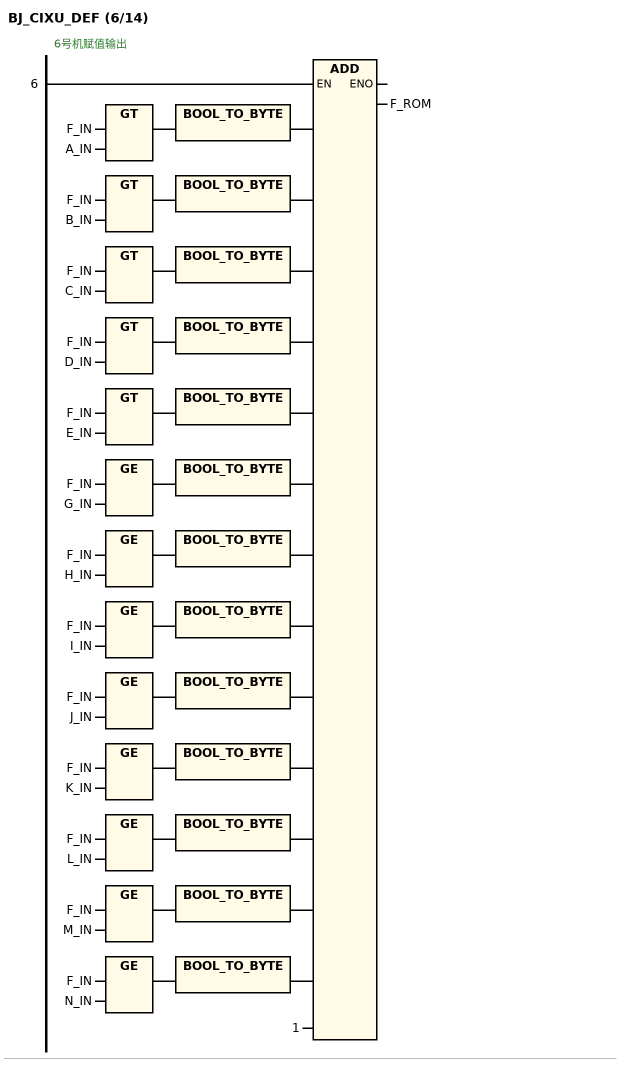
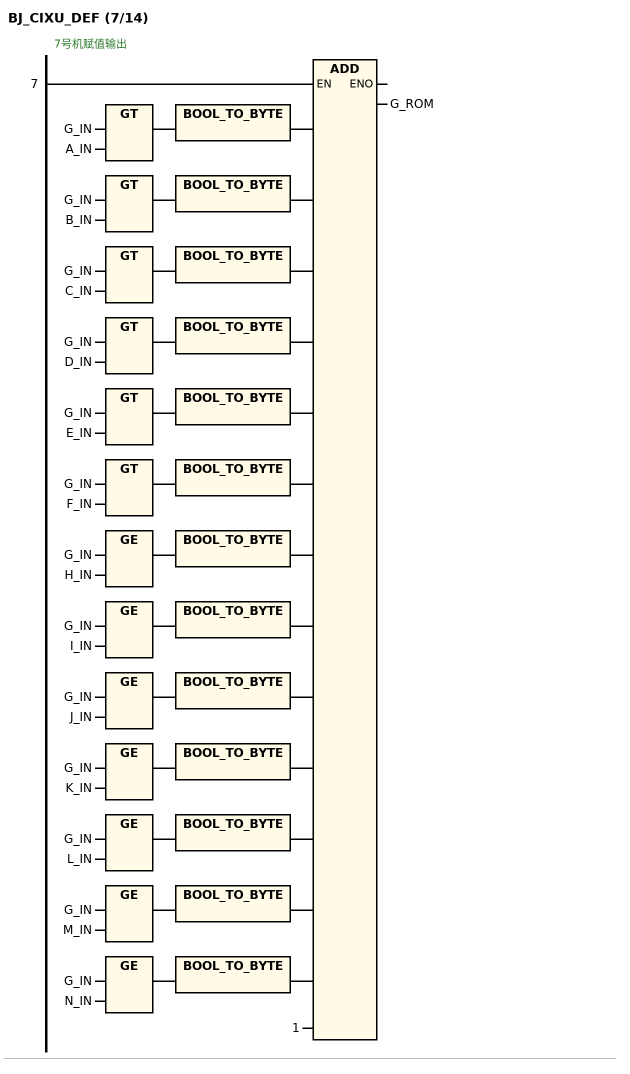
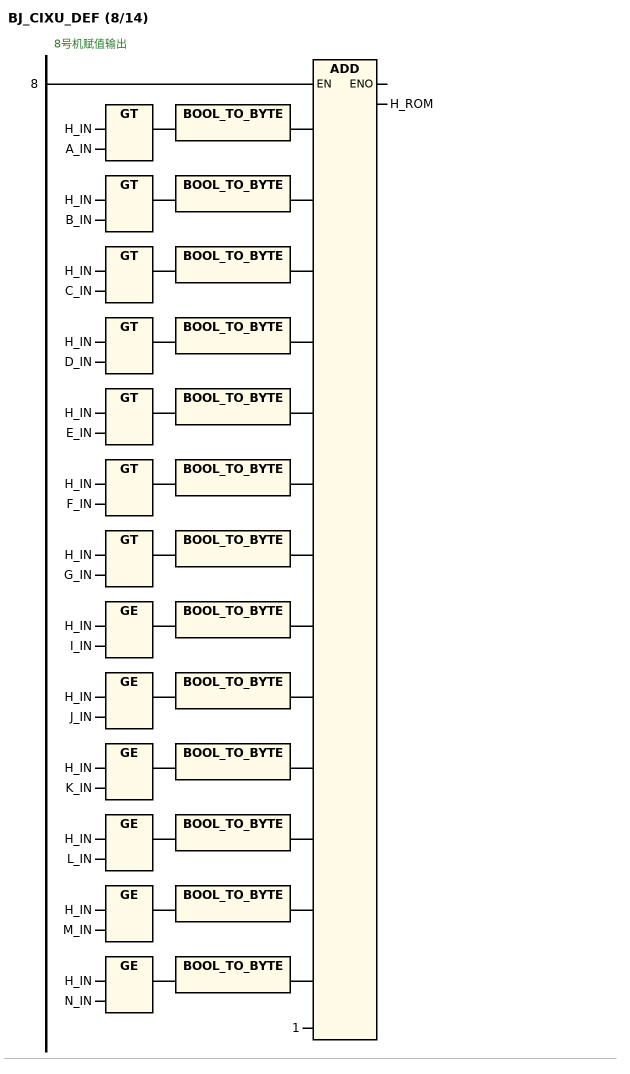
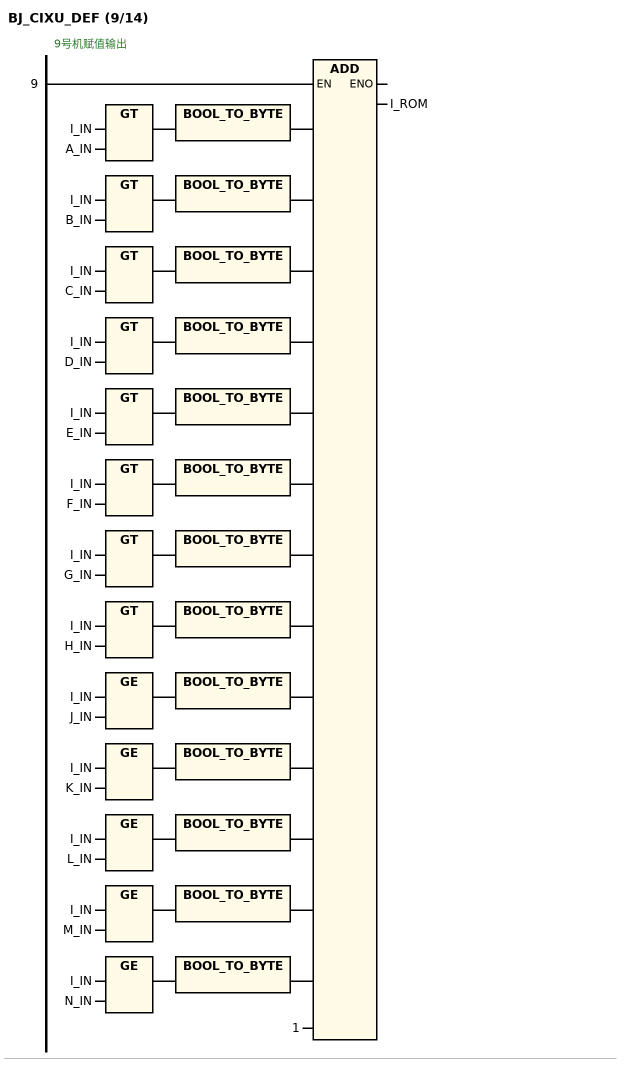
